FUNCTION_BLOCK FB_Integer_Out
VAR_INPUT
END_VAR
VAR_IN_OUT
	Input1																: INT;
	Input2																: INT;
END_VAR
VAR
	Last1																: INT;
	Last2																: INT;
END_VAR

// Theseus - FB_Integer_Out
// Rev 1.0 - April 24, 2024

IF Input2 <> Last2 THEN
	Last2																:= Input2;
	Input1																:= Input2;
	Last1																:= Input2;
ELSIF Input1 <> Last1 THEN
	Last1																:= Input1;
	Input2																:= Input1;
	Last2																:= Input1;
END_IF

END_FUNCTION_BLOCK

(* stored: Version 1.1.0.1, ProductVersion 3.1.4024.12
   POU FB_Integer_Out: Id {1b4126e1-3c47-44e5-aa10-ef4647bf40e4}, SpecialFunc None *)
